# EPICS autosave request: iocBoot/iocSaveEnergy/auto_settings.req
file "saveEnergy_settings.req", P=$(P), R=$(R)
